// TIA Portal V20 export
TYPE "typeRollChangeMode"
// stored: Access Published, IsFailsafeCompliant true, Namespace Safety
   STRUCT
      Auto : Bool;
      RollChange : Bool;
   END_STRUCT;
END_TYPE
